PROGRAM MAIN
VAR
	runOnlyOnce : BOOL := FALSE;
END_VAR

IF NOT runOnlyOnce THEN
ADSLOGSTR(msgCtrlMask := ADSLOG_MSGTYPE_ERROR OR ADSLOG_MSGTYPE_LOG, msgFmtStr := 'Hello World',strArg := '');
	runOnlyOnce := TRUE;
	END_IF

END_PROGRAM

(* stored: Version 1.1.0.1, ProductVersion 3.1.4024.12
   POU MAIN: Id {375d9c5e-2873-48ed-9862-cd3470397a2c}, SpecialFunc None *)
